FUNCTION RGBWtoINT : INT
VAR_INPUT
END_VAR
VAR
END_VAR

END_FUNCTION

(* stored: Version 1.1.0.1, ProductVersion 3.1.4024.12
   POU RGBWtoINT: Id {0750f7b7-a3ac-47d5-a092-a91a39eece94}, SpecialFunc None *)
